PROGRAM Pumps
VAR
	Pump_1 : Pump;
END_VAR
VAR // added by the converter: edge detectors and wires of the graphical bodies
    _w1, _w2, _w3, _w4, _w5, _w6 : BOOL;
END_VAR

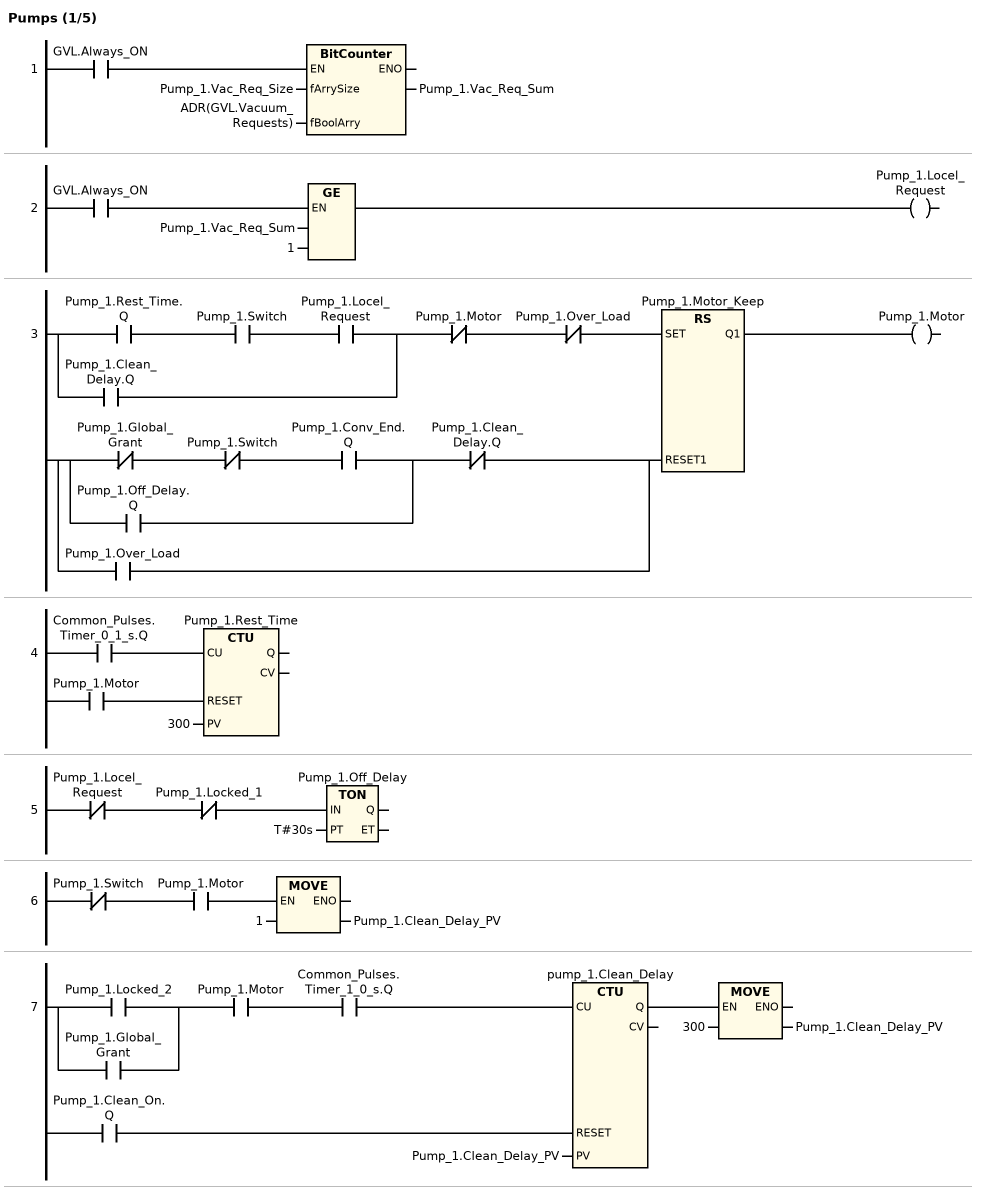
// NETWORK 1
IF GVL.Always_ON THEN
    Pump_1.Vac_Req_Sum := BitCounter(fArrySize := Pump_1.Vac_Req_Size, fBoolArry := ADR(GVL.Vacuum_Requests));
END_IF

// NETWORK 2
Pump_1.Locel_Request := GVL.Always_ON AND Pump_1.Vac_Req_Sum >= 1;

// NETWORK 3
Pump_1.Motor_Keep(SET := (Pump_1.Rest_Time.Q AND Pump_1.Switch AND Pump_1.Locel_Request OR Pump_1.Clean_Delay.Q) AND NOT Pump_1.Motor AND NOT Pump_1.Over_Load, RESET1 := (NOT Pump_1.Global_Grant AND NOT Pump_1.Switch AND Pump_1.Conv_End.Q OR Pump_1.Off_Delay.Q) AND NOT Pump_1.Clean_Delay.Q OR Pump_1.Over_Load); // RS
Pump_1.Motor := Pump_1.Motor_Keep.Q1;

// NETWORK 4
Pump_1.Rest_Time(CU := Common_Pulses.Timer_0_1_s.Q, RESET := Pump_1.Motor, PV := 300); // CTU

// NETWORK 5
Pump_1.Off_Delay(IN := NOT Pump_1.Locel_Request AND NOT Pump_1.Locked_1, PT := T#30s); // TON

// NETWORK 6
IF NOT Pump_1.Switch AND Pump_1.Motor THEN Pump_1.Clean_Delay_PV := 1; END_IF

// NETWORK 7
pump_1.Clean_Delay(
    CU := (Pump_1.Locked_2 OR Pump_1.Global_Grant) AND Pump_1.Motor AND Common_Pulses.Timer_1_0_s.Q,
    RESET := Pump_1.Clean_On.Q,
    PV := Pump_1.Clean_Delay_PV); // CTU
IF pump_1.Clean_Delay.Q THEN Pump_1.Clean_Delay_PV := 300; END_IF

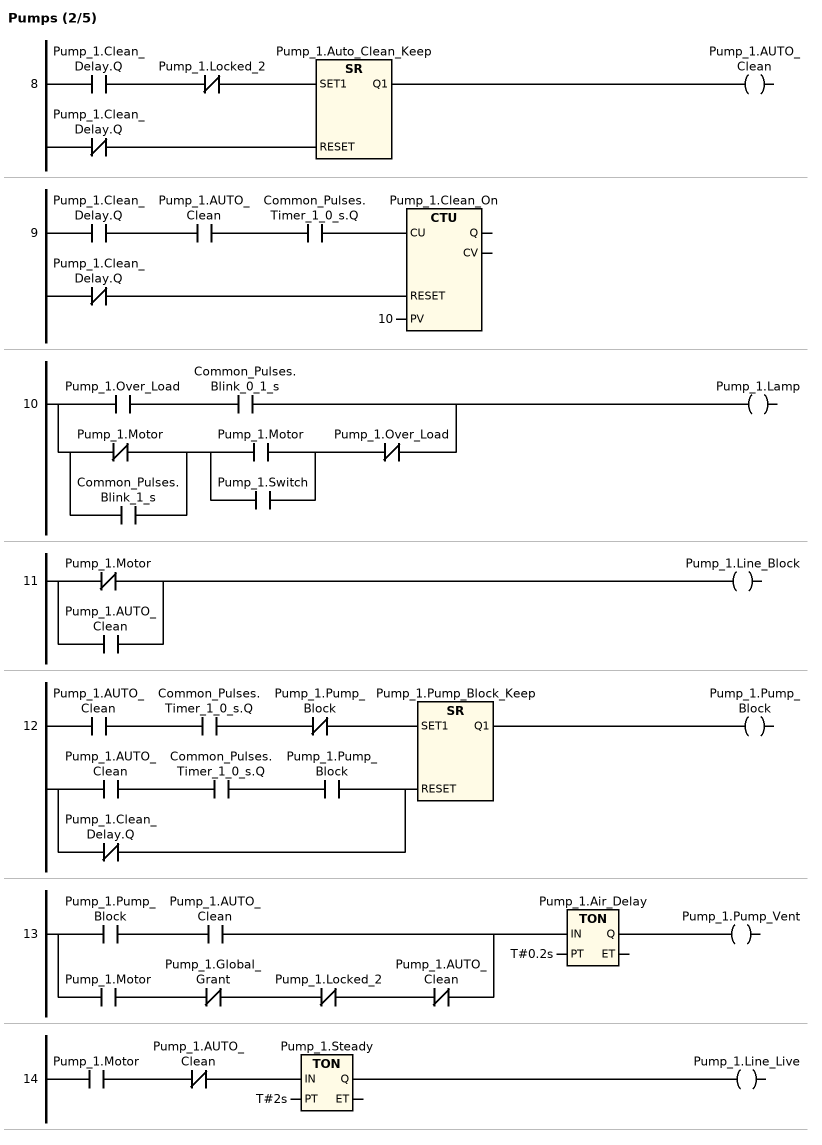
// NETWORK 8
Pump_1.Auto_Clean_Keep(SET1 := Pump_1.Clean_Delay.Q AND NOT Pump_1.Locked_2, RESET := NOT Pump_1.Clean_Delay.Q); // SR
Pump_1.AUTO_Clean := Pump_1.Auto_Clean_Keep.Q1;

// NETWORK 9
Pump_1.Clean_On(
    CU := Pump_1.Clean_Delay.Q AND Pump_1.AUTO_Clean AND Common_Pulses.Timer_1_0_s.Q,
    RESET := NOT Pump_1.Clean_Delay.Q,
    PV := 10); // CTU

// NETWORK 10
Pump_1.Lamp := Pump_1.Over_Load AND Common_Pulses.Blink_0_1_s OR (NOT Pump_1.Motor OR Common_Pulses.Blink_1_s) AND (Pump_1.Motor OR Pump_1.Switch) AND NOT Pump_1.Over_Load;

// NETWORK 11
Pump_1.Line_Block := NOT Pump_1.Motor OR Pump_1.AUTO_Clean;

// NETWORK 12
Pump_1.Pump_Block_Keep(SET1 := Pump_1.AUTO_Clean AND Common_Pulses.Timer_1_0_s.Q AND NOT Pump_1.Pump_Block, RESET := Pump_1.AUTO_Clean AND Common_Pulses.Timer_1_0_s.Q AND Pump_1.Pump_Block OR NOT Pump_1.Clean_Delay.Q); // SR
Pump_1.Pump_Block := Pump_1.Pump_Block_Keep.Q1;

// NETWORK 13
Pump_1.Air_Delay(IN := Pump_1.Pump_Block AND Pump_1.AUTO_Clean OR Pump_1.Motor AND NOT Pump_1.Global_Grant AND NOT Pump_1.Locked_2 AND NOT Pump_1.AUTO_Clean, PT := T#0.2s); // TON
Pump_1.Pump_Vent := Pump_1.Air_Delay.Q;

// NETWORK 14
Pump_1.Steady(IN := Pump_1.Motor AND NOT Pump_1.AUTO_Clean, PT := T#2s); // TON
Pump_1.Line_Live := Pump_1.Steady.Q;

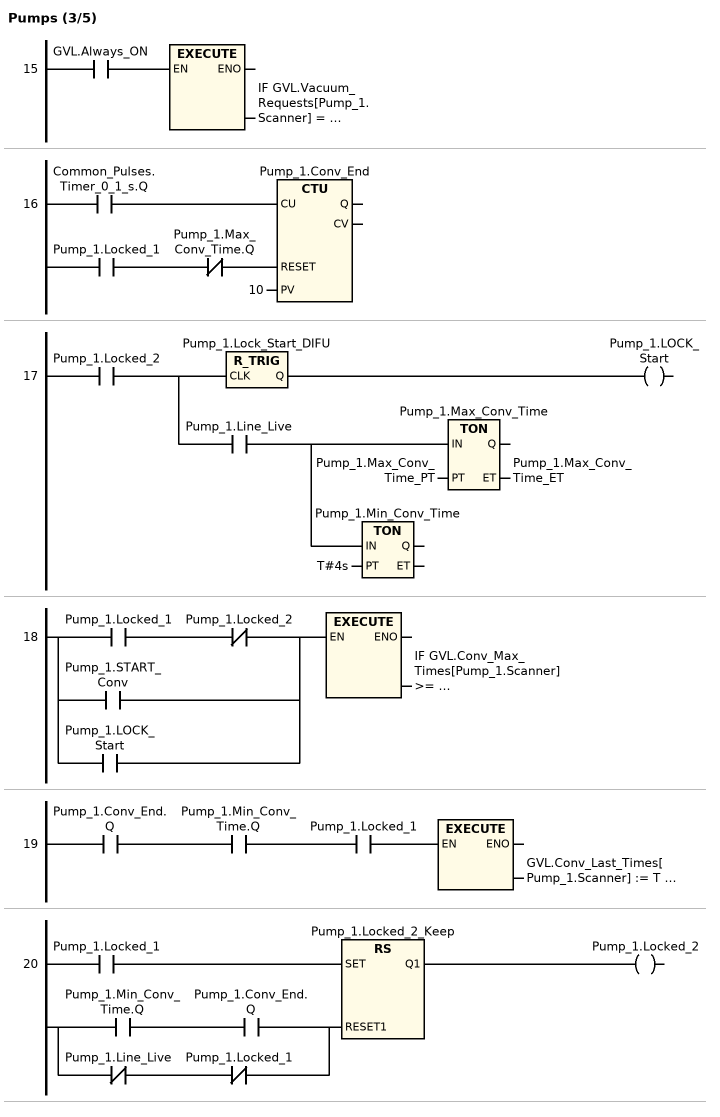
// NETWORK 15
IF GVL.Always_ON THEN
    IF GVL.Vacuum_Requests[Pump_1.Scanner] = 1 THEN 
    	Pump_1.Locked_1 := TRUE;
    	ELSE Pump_1.Locked_1 := FALSE;
    END_IF
END_IF

// NETWORK 16
Pump_1.Conv_End(
    CU := Common_Pulses.Timer_0_1_s.Q,
    RESET := Pump_1.Locked_1 AND NOT Pump_1.Max_Conv_Time.Q,
    PV := 10); // CTU

// NETWORK 17
Pump_1.Lock_Start_DIFU(CLK := Pump_1.Locked_2); // R_TRIG
Pump_1.LOCK_Start := Pump_1.Lock_Start_DIFU.Q;
_w1 := Pump_1.Locked_2 AND Pump_1.Line_Live;
Pump_1.Max_Conv_Time(IN := _w1, PT := Pump_1.Max_Conv_Time_PT, ET => Pump_1.Max_Conv_Time_ET); // TON
Pump_1.Min_Conv_Time(IN := _w1, PT := T#4s); // TON

// NETWORK 18
IF Pump_1.Locked_1 AND NOT Pump_1.Locked_2 OR Pump_1.START_Conv OR Pump_1.LOCK_Start THEN
    IF GVL.Conv_Max_Times[Pump_1.Scanner] >= 5000 THEN
    	Pump_1.Max_Conv_Time_PT := DWORD_TO_TIME(GVL.Conv_Max_Times[Pump_1.Scanner]);
    	ELSE Pump_1.Max_Conv_Time.PT := T#5S;
    END_IF
END_IF

// NETWORK 19
IF Pump_1.Conv_End.Q AND Pump_1.Min_Conv_Time.Q AND Pump_1.Locked_1 THEN
    GVL.Conv_Last_Times[Pump_1.Scanner] := TIME_TO_DWORD(Pump_1.Max_Conv_Time.ET);
    MEMSET (destAddr := ADR(GVL.Vacuum_Requests), fillByte := 0, n := SIZEOF(GVL.Vacuum_Requests));
END_IF

// NETWORK 20
Pump_1.Locked_2_Keep(SET := Pump_1.Locked_1, RESET1 := Pump_1.Min_Conv_Time.Q AND Pump_1.Conv_End.Q OR NOT Pump_1.Line_Live AND NOT Pump_1.Locked_1); // RS
Pump_1.Locked_2 := Pump_1.Locked_2_Keep.Q1;

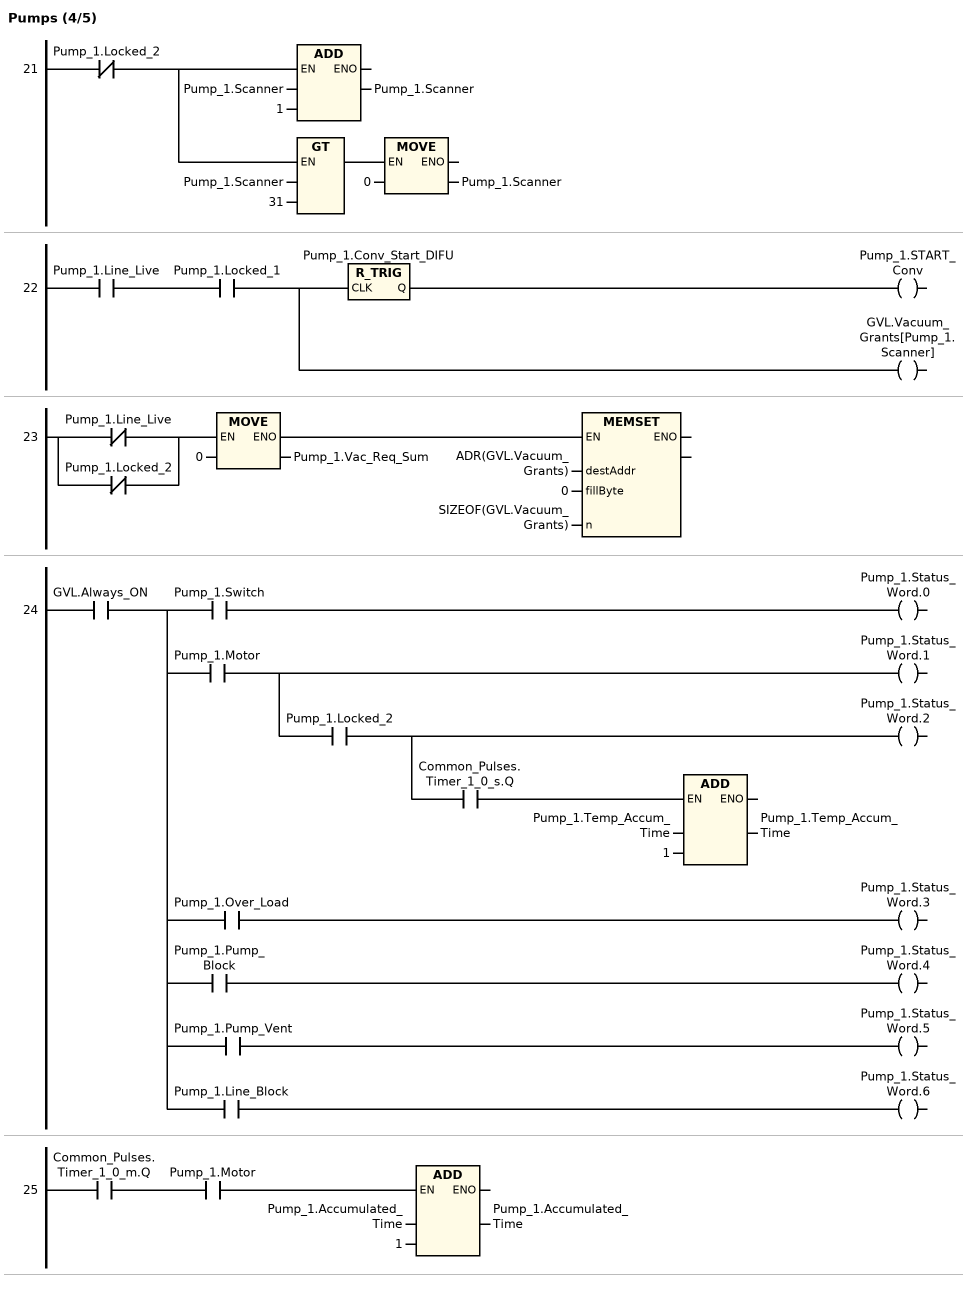
// NETWORK 21
_w2 := NOT Pump_1.Locked_2;
IF _w2 THEN Pump_1.Scanner := Pump_1.Scanner + 1; END_IF
IF _w2 AND Pump_1.Scanner > 31 THEN Pump_1.Scanner := 0; END_IF

// NETWORK 22
_w3 := Pump_1.Line_Live AND Pump_1.Locked_1;
Pump_1.Conv_Start_DIFU(CLK := _w3); // R_TRIG
Pump_1.START_Conv := Pump_1.Conv_Start_DIFU.Q;
GVL.Vacuum_Grants[Pump_1.Scanner] := _w3;

// NETWORK 23
_w4 := NOT Pump_1.Line_Live OR NOT Pump_1.Locked_2;
IF _w4 THEN Pump_1.Vac_Req_Sum := 0; END_IF
IF _w4 THEN MEMSET(destAddr := ADR(GVL.Vacuum_Grants), fillByte := 0, n := SIZEOF(GVL.Vacuum_Grants)); END_IF

// NETWORK 24
Pump_1.Status_Word.0 := GVL.Always_ON AND Pump_1.Switch;
_w5 := GVL.Always_ON AND Pump_1.Motor;
Pump_1.Status_Word.1 := _w5;
_w6 := _w5 AND Pump_1.Locked_2;
Pump_1.Status_Word.2 := _w6;
IF _w6 AND Common_Pulses.Timer_1_0_s.Q THEN Pump_1.Temp_Accum_Time := Pump_1.Temp_Accum_Time + 1; END_IF
Pump_1.Status_Word.3 := GVL.Always_ON AND Pump_1.Over_Load;
Pump_1.Status_Word.4 := GVL.Always_ON AND Pump_1.Pump_Block;
Pump_1.Status_Word.5 := GVL.Always_ON AND Pump_1.Pump_Vent;
Pump_1.Status_Word.6 := GVL.Always_ON AND Pump_1.Line_Block;

// NETWORK 25
IF Common_Pulses.Timer_1_0_m.Q AND Pump_1.Motor THEN Pump_1.Accumulated_Time := Pump_1.Accumulated_Time + 1; END_IF

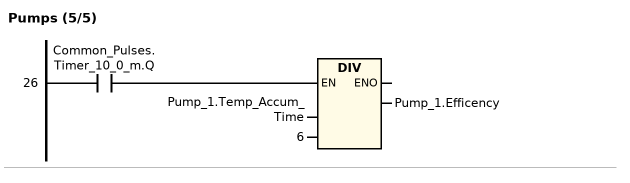
// NETWORK 26
IF Common_Pulses.Timer_10_0_m.Q THEN Pump_1.Efficency := Pump_1.Temp_Accum_Time / 6; END_IF

END_PROGRAM

(* stored: Version 1.1.0.1, ProductVersion 3.1.4024.13
   POU Pumps: Id {159c9f79-2307-412c-9ac7-43880167eddb}, SpecialFunc None *)
